//=============================================================================
// ST10_Flow22_JMagnetLifting.scl
// 1:1 CONVERSION FROM TIA PORTAL V18 GRAPH XML
// Generated: 2026-02-02
//=============================================================================

TYPE
    E_STEP_ST10_Flow22_JMagnetLifting : (
        STEP_ST10_Flow22_JMagnetLifting_WaitingPalletUnloading := 135,
        STEP_ST10_Flow22_JMagnetLifting_S3 := 3,
        STEP_ST10_Flow22_JMagnetLifting_TimeDelay := 22,
        STEP_ST10_Flow22_JMagnetLifting_J_magnetLiftingPalletLocationCylindertoHP := 129,
        STEP_ST10_Flow22_JMagnetLifting_Process_Finish := 237,
        STEP_ST10_Flow22_JMagnetLifting_F22_Initial := 1,
        STEP_ST10_Flow22_JMagnetLifting_S4 := 4,
        STEP_ST10_Flow22_JMagnetLifting_PalletRequest := 136,
        STEP_ST10_Flow22_JMagnetLifting_WaitRobotInitialFinish := 8,
        STEP_ST10_Flow22_JMagnetLifting_MotorCWStart := 24,
        STEP_ST10_Flow22_JMagnetLifting_J_magnetLiftingPalletLocationCylindertoHP_3 := 139,
        STEP_ST10_Flow22_JMagnetLifting_S2 := 2,
        STEP_ST10_Flow22_JMagnetLifting_RequestRobotPickPallet := 134,
        STEP_ST10_Flow22_JMagnetLifting_StatusError := 20,
        STEP_ST10_Flow22_JMagnetLifting_MotorCCWRun_1 := 144,
        STEP_ST10_Flow22_JMagnetLifting_CheckStopPalletExist := 21,
        STEP_ST10_Flow22_JMagnetLifting_MotorCCWStart := 23,
        STEP_ST10_Flow22_JMagnetLifting_S10_InitialFinish := 10,
        STEP_ST10_Flow22_JMagnetLifting_WaitRobotTaskFinish := 145,
        STEP_ST10_Flow22_JMagnetLifting_RobotCountClear0 := 137,
        STEP_ST10_Flow22_JMagnetLifting_MotorCCWRun := 140,
        STEP_ST10_Flow22_JMagnetLifting_J_magnetLiftingPalletLocationCylindertoHP_2 := 138,
        STEP_ST10_Flow22_JMagnetLifting_H_shaftLiftingLiftingCylinderToWP := 116,
        STEP_ST10_Flow22_JMagnetLifting_CheckPalletExist := 133,
        STEP_ST10_Flow22_JMagnetLifting_J_magnetLiftingPalletLocationCylindertoWP_1 := 130,
        STEP_ST10_Flow22_JMagnetLifting_Step131 := 131,
        STEP_ST10_Flow22_JMagnetLifting_CheckShaftLiftingCylinderPos := 117,
        STEP_ST10_Flow22_JMagnetLifting_J_magnetLiftingPalletLocationCylindertoHP_4 := 143,
        STEP_ST10_Flow22_JMagnetLifting_ProcessStart := 100,
        STEP_ST10_Flow22_JMagnetLifting_MotorStop := 132,
        STEP_ST10_Flow22_JMagnetLifting_Motor_Stop := 141,
        STEP_ST10_Flow22_JMagnetLifting_J_magnetLiftingCylinderToWP := 142,
        STEP_ST10_Flow22_JMagnetLifting_S5_MESInitial := 5,
    ) INT := 1;
END_TYPE

CONST
    STEP_ST10_Flow22_JMagnetLifting_WaitingPalletUnloading := 135;
    STEP_ST10_Flow22_JMagnetLifting_S3 := 3;
    STEP_ST10_Flow22_JMagnetLifting_TimeDelay := 22;
    STEP_ST10_Flow22_JMagnetLifting_J_magnetLiftingPalletLocationCylindertoHP := 129;
    STEP_ST10_Flow22_JMagnetLifting_Process_Finish := 237;
    STEP_ST10_Flow22_JMagnetLifting_F22_Initial := 1;
    STEP_ST10_Flow22_JMagnetLifting_S4 := 4;
    STEP_ST10_Flow22_JMagnetLifting_PalletRequest := 136;
    STEP_ST10_Flow22_JMagnetLifting_WaitRobotInitialFinish := 8;
    STEP_ST10_Flow22_JMagnetLifting_MotorCWStart := 24;
    STEP_ST10_Flow22_JMagnetLifting_J_magnetLiftingPalletLocationCylindertoHP_3 := 139;
    STEP_ST10_Flow22_JMagnetLifting_S2 := 2;
    STEP_ST10_Flow22_JMagnetLifting_RequestRobotPickPallet := 134;
    STEP_ST10_Flow22_JMagnetLifting_StatusError := 20;
    STEP_ST10_Flow22_JMagnetLifting_MotorCCWRun_1 := 144;
    STEP_ST10_Flow22_JMagnetLifting_CheckStopPalletExist := 21;
    STEP_ST10_Flow22_JMagnetLifting_MotorCCWStart := 23;
    STEP_ST10_Flow22_JMagnetLifting_S10_InitialFinish := 10;
    STEP_ST10_Flow22_JMagnetLifting_WaitRobotTaskFinish := 145;
    STEP_ST10_Flow22_JMagnetLifting_RobotCountClear0 := 137;
    STEP_ST10_Flow22_JMagnetLifting_MotorCCWRun := 140;
    STEP_ST10_Flow22_JMagnetLifting_J_magnetLiftingPalletLocationCylindertoHP_2 := 138;
    STEP_ST10_Flow22_JMagnetLifting_H_shaftLiftingLiftingCylinderToWP := 116;
    STEP_ST10_Flow22_JMagnetLifting_CheckPalletExist := 133;
    STEP_ST10_Flow22_JMagnetLifting_J_magnetLiftingPalletLocationCylindertoWP_1 := 130;
    STEP_ST10_Flow22_JMagnetLifting_Step131 := 131;
    STEP_ST10_Flow22_JMagnetLifting_CheckShaftLiftingCylinderPos := 117;
    STEP_ST10_Flow22_JMagnetLifting_J_magnetLiftingPalletLocationCylindertoHP_4 := 143;
    STEP_ST10_Flow22_JMagnetLifting_ProcessStart := 100;
    STEP_ST10_Flow22_JMagnetLifting_MotorStop := 132;
    STEP_ST10_Flow22_JMagnetLifting_Motor_Stop := 141;
    STEP_ST10_Flow22_JMagnetLifting_J_magnetLiftingCylinderToWP := 142;
    STEP_ST10_Flow22_JMagnetLifting_S5_MESInitial := 5;
END_CONST

FUNCTION_BLOCK "ST10_Flow22_JMagnetLifting_1to1"
{ S7_Optimized_Access := 'TRUE' }
VERSION : 1.0

VAR_INPUT
    iSysInface : "RCS_SysComInterface_V1";
END_VAR

VAR_IN_OUT
    ioPM_Inface : "RCS_PMInterface_V1";
    ioStatus : Int;
END_VAR

VAR_OUTPUT
    oAlarmID : Int;
END_VAR

VAR
    State : INT := 1;
    act_InitialRun : Bool;
    act_InitialOK : Bool;
    act_WaitRunning : Bool;
    act_Running : Bool;
    act_ProcessComplete : Bool;
    act_ProcessStart : Bool;
    act_UnPause : Bool;
    bError : Bool;
    wErrorID : Word;
END_VAR

BEGIN
    //======================================================================
    // STATE MACHINE - Inline Transition Conditions
    //======================================================================

    CASE #State OF

        // ===========================================
        // STEP 135: WaitingPalletUnloading
        // ===========================================
        STEP_ST10_Flow22_JMagnetLifting_WaitingPalletUnloading:
            // No actions in XML

            // Transition to next step: 3
            IF TRUE THEN  // Sequential transition - review XML for actual condition
                #State := STEP_ST10_Flow22_JMagnetLifting_S3;
            END_IF;

        // ===========================================
        // STEP 3: S3
        // ===========================================
        STEP_ST10_Flow22_JMagnetLifting_S3:
            // No actions in XML

            // Transition to next step: 22
            IF TRUE THEN  // Sequential transition - review XML for actual condition
                #State := STEP_ST10_Flow22_JMagnetLifting_TimeDelay;
            END_IF;

        // ===========================================
        // STEP 22: TimeDelay
        // ===========================================
        STEP_ST10_Flow22_JMagnetLifting_TimeDelay:
            // No actions in XML

            // Transition to next step: 129
            IF TRUE THEN  // Sequential transition - review XML for actual condition
                #State := STEP_ST10_Flow22_JMagnetLifting_J_magnetLiftingPalletLocationCylindertoHP;
            END_IF;

        // ===========================================
        // STEP 129: J-magnetLiftingPalletLocationCylindertoHP
        // ===========================================
        STEP_ST10_Flow22_JMagnetLifting_J_magnetLiftingPalletLocationCylindertoHP:
            // Action Qualifier=S
            // Token: "ST10Cylinder".Cy[32].Inout.AutoGoHome
            "ST10Cylinder".Cy[32].Inout.AutoGoHome := TRUE;
            // Action Qualifier=R
            // Token: "ST10Cylinder".Cy[32].Inout.AutoGoWork
            "ST10Cylinder".Cy[32].Inout.AutoGoWork := FALSE;

            // Transition to next step: 237
            IF TRUE THEN  // Sequential transition - review XML for actual condition
                #State := STEP_ST10_Flow22_JMagnetLifting_Process_Finish;
            END_IF;

        // ===========================================
        // STEP 237: Process Finish
        // ===========================================
        STEP_ST10_Flow22_JMagnetLifting_Process_Finish:
            // No actions in XML

            // Transition to next step: 1
            IF TRUE THEN  // Sequential transition - review XML for actual condition
                #State := STEP_ST10_Flow22_JMagnetLifting_F22_Initial;
            END_IF;

        // ===========================================
        // STEP 1: F22_Initial
        // ===========================================
        STEP_ST10_Flow22_JMagnetLifting_F22_Initial:
            // Action Qualifier=S
            // Token: #ioPM_Inface.InitialRun
            #ioPM_Inface.InitialRun := TRUE;
            // Action Qualifier=R
            // Token: #ioPM_Inface.InitialOK
            #ioPM_Inface.InitialOK := FALSE;
            // Action Qualifier=R
            // Token: #ioPM_Inface.WaitRunning
            #ioPM_Inface.WaitRunning := FALSE;
            // Action Qualifier=R
            // Token: #ioPM_Inface.Running
            #ioPM_Inface.Running := FALSE;
            // Action Qualifier=R
            // Token: #ioPM_Inface.ProcessComplete
            #ioPM_Inface.ProcessComplete := FALSE;
            // Action Qualifier=R
            // Token: #ioPM_Inface.UnPause
            #ioPM_Inface.UnPause := FALSE;
            // Action Qualifier=R
            // Token: "Station_Sys".Cmd.Calibration
            "Station_Sys".Cmd.Calibration := FALSE;
            // Action Qualifier=R
            // Token: "Station_Sys".Cmd.ChangeOver
            "Station_Sys".Cmd.ChangeOver := FALSE;
            // Action Qualifier=N
            // Token: //"ST350_Sys".Cmd.DryRun
            //"ST350_Sys".Cmd.DryRun;
            // Action Qualifier=R
            // Token: "Station_Sys".Cmd.Reserve
            "Station_Sys".Cmd.Reserve := FALSE;
            // Action Qualifier=R
            // Token: "Station_Sys".Cmd.OneCycle
            "Station_Sys".Cmd.OneCycle := FALSE;

            // Transition to next step: 4
            IF TRUE THEN  // Sequential transition - review XML for actual condition
                #State := STEP_ST10_Flow22_JMagnetLifting_S4;
            END_IF;

        // ===========================================
        // STEP 4: S4
        // ===========================================
        STEP_ST10_Flow22_JMagnetLifting_S4:
            // No actions in XML

            // Transition to next step: 136
            IF TRUE THEN  // Sequential transition - review XML for actual condition
                #State := STEP_ST10_Flow22_JMagnetLifting_PalletRequest;
            END_IF;

        // ===========================================
        // STEP 136: PalletRequest
        // ===========================================
        STEP_ST10_Flow22_JMagnetLifting_PalletRequest:
            // Action Qualifier=N
            // Token: "AutoProcessControl".Global.J.LoadStopRequestPallet_4
            "AutoProcessControl".Global.J.LoadStopRequestPallet_4;

            // Transition to next step: 8
            IF TRUE THEN  // Sequential transition - review XML for actual condition
                #State := STEP_ST10_Flow22_JMagnetLifting_WaitRobotInitialFinish;
            END_IF;

        // ===========================================
        // STEP 8: WaitRobotInitialFinish
        // ===========================================
        STEP_ST10_Flow22_JMagnetLifting_WaitRobotInitialFinish:
            // No actions in XML

            // Transition to next step: 24
            IF TRUE THEN  // Sequential transition - review XML for actual condition
                #State := STEP_ST10_Flow22_JMagnetLifting_MotorCWStart;
            END_IF;

        // ===========================================
        // STEP 24: MotorCWStart
        // ===========================================
        STEP_ST10_Flow22_JMagnetLifting_MotorCWStart:
            // Action Qualifier=R
            // Token: "MotorControl".Dev[2].Auto.CCWStart
            "MotorControl".Dev[2].Auto.CCWStart := FALSE;
            // Action Qualifier=S
            // Token: "MotorControl".Dev[2].Auto.Start
            "MotorControl".Dev[2].Auto.Start := TRUE;

            // Transition to next step: 139
            IF TRUE THEN  // Sequential transition - review XML for actual condition
                #State := STEP_ST10_Flow22_JMagnetLifting_J_magnetLiftingPalletLocationCylindertoHP_3;
            END_IF;

        // ===========================================
        // STEP 139: J-magnetLiftingPalletLocationCylindertoHP_3
        // ===========================================
        STEP_ST10_Flow22_JMagnetLifting_J_magnetLiftingPalletLocationCylindertoHP_3:
            // Action Qualifier=S
            // Token: "ST10Cylinder".Cy[31].Inout.AutoGoHome
            "ST10Cylinder".Cy[31].Inout.AutoGoHome := TRUE;
            // Action Qualifier=R
            // Token: "ST10Cylinder".Cy[31].Inout.AutoGoWork
            "ST10Cylinder".Cy[31].Inout.AutoGoWork := FALSE;

            // Transition to next step: 2
            IF TRUE THEN  // Sequential transition - review XML for actual condition
                #State := STEP_ST10_Flow22_JMagnetLifting_S2;
            END_IF;

        // ===========================================
        // STEP 2: S2
        // ===========================================
        STEP_ST10_Flow22_JMagnetLifting_S2:
            // No actions in XML

            // Transition to next step: 134
            IF TRUE THEN  // Sequential transition - review XML for actual condition
                #State := STEP_ST10_Flow22_JMagnetLifting_RequestRobotPickPallet;
            END_IF;

        // ===========================================
        // STEP 134: RequestRobotPickPallet
        // ===========================================
        STEP_ST10_Flow22_JMagnetLifting_RequestRobotPickPallet:
            // Action Qualifier=N
            // Token: "AutoProcessControl".J_MagnetLine.Robot2PickPrimit
            "AutoProcessControl".J_MagnetLine.Robot2PickPrimit;

            // Transition to next step: 20
            IF TRUE THEN  // Sequential transition - review XML for actual condition
                #State := STEP_ST10_Flow22_JMagnetLifting_StatusError;
            END_IF;

        // ===========================================
        // STEP 20: StatusError
        // ===========================================
        STEP_ST10_Flow22_JMagnetLifting_StatusError:
            // Action Qualifier=S
            // Token: "ST10_DeviceError".J.MagnetLine.LiftingCylStatusError
            "ST10_DeviceError".J.MagnetLine.LiftingCylStatusError := TRUE;

            // Transition to next step: 144
            IF TRUE THEN  // Sequential transition - review XML for actual condition
                #State := STEP_ST10_Flow22_JMagnetLifting_MotorCCWRun_1;
            END_IF;

        // ===========================================
        // STEP 144: MotorCCWRun_1
        // ===========================================
        STEP_ST10_Flow22_JMagnetLifting_MotorCCWRun_1:
            // Action Qualifier=S
            // Token: "MotorControl".Dev[2].Auto.CCWStart
            "MotorControl".Dev[2].Auto.CCWStart := TRUE;
            // Action Qualifier=S
            // Token: "MotorControl".Dev[2].Auto.Start
            "MotorControl".Dev[2].Auto.Start := TRUE;

            // Transition to next step: 21
            IF TRUE THEN  // Sequential transition - review XML for actual condition
                #State := STEP_ST10_Flow22_JMagnetLifting_CheckStopPalletExist;
            END_IF;

        // ===========================================
        // STEP 21: CheckStopPalletExist
        // ===========================================
        STEP_ST10_Flow22_JMagnetLifting_CheckStopPalletExist:
            // No actions in XML

            // Transition to next step: 23
            IF TRUE THEN  // Sequential transition - review XML for actual condition
                #State := STEP_ST10_Flow22_JMagnetLifting_MotorCCWStart;
            END_IF;

        // ===========================================
        // STEP 23: MotorCCWStart
        // ===========================================
        STEP_ST10_Flow22_JMagnetLifting_MotorCCWStart:
            // Action Qualifier=S
            // Token: "MotorControl".Dev[2].Auto.CCWStart
            "MotorControl".Dev[2].Auto.CCWStart := TRUE;
            // Action Qualifier=S
            // Token: "MotorControl".Dev[2].Auto.Start
            "MotorControl".Dev[2].Auto.Start := TRUE;

            // Transition to next step: 10
            IF TRUE THEN  // Sequential transition - review XML for actual condition
                #State := STEP_ST10_Flow22_JMagnetLifting_S10_InitialFinish;
            END_IF;

        // ===========================================
        // STEP 10: S10_InitialFinish
        // ===========================================
        STEP_ST10_Flow22_JMagnetLifting_S10_InitialFinish:
            // Action Qualifier=S
            // Token: #ioPM_Inface.InitialOK
            #ioPM_Inface.InitialOK := TRUE;

            // Transition to next step: 145
            IF TRUE THEN  // Sequential transition - review XML for actual condition
                #State := STEP_ST10_Flow22_JMagnetLifting_WaitRobotTaskFinish;
            END_IF;

        // ===========================================
        // STEP 145: WaitRobotTaskFinish
        // ===========================================
        STEP_ST10_Flow22_JMagnetLifting_WaitRobotTaskFinish:
            // No actions in XML

            // Transition to next step: 137
            IF TRUE THEN  // Sequential transition - review XML for actual condition
                #State := STEP_ST10_Flow22_JMagnetLifting_RobotCountClear0;
            END_IF;

        // ===========================================
        // STEP 137: RobotCountClear0
        // ===========================================
        STEP_ST10_Flow22_JMagnetLifting_RobotCountClear0:
            // Action Qualifier=N
            // Token: "KukaRobot2_CtrlDB".sPLCtoROB.User.Cycle.DI242_NewPallet
            "KukaRobot2_CtrlDB".sPLCtoROB.User.Cycle.DI242_NewPallet;
            // Action Qualifier=R
            // Token: "MotorControl".Dev[2].Auto.Start
            "MotorControl".Dev[2].Auto.Start := FALSE;

            // Transition to next step: 140
            IF TRUE THEN  // Sequential transition - review XML for actual condition
                #State := STEP_ST10_Flow22_JMagnetLifting_MotorCCWRun;
            END_IF;

        // ===========================================
        // STEP 140: MotorCCWRun
        // ===========================================
        STEP_ST10_Flow22_JMagnetLifting_MotorCCWRun:
            // Action Qualifier=S
            // Token: "MotorControl".Dev[2].Auto.CCWStart
            "MotorControl".Dev[2].Auto.CCWStart := TRUE;
            // Action Qualifier=S
            // Token: "MotorControl".Dev[2].Auto.Start
            "MotorControl".Dev[2].Auto.Start := TRUE;
            // Action Qualifier=R
            // Token: "MotorControl".Dev[14].Auto.CCWStart
            "MotorControl".Dev[14].Auto.CCWStart := FALSE;
            // Action Qualifier=S
            // Token: "MotorControl".Dev[14].Auto.Start
            "MotorControl".Dev[14].Auto.Start := TRUE;

            // Transition to next step: 138
            IF TRUE THEN  // Sequential transition - review XML for actual condition
                #State := STEP_ST10_Flow22_JMagnetLifting_J_magnetLiftingPalletLocationCylindertoHP_2;
            END_IF;

        // ===========================================
        // STEP 138: J-magnetLiftingPalletLocationCylindertoHP_2
        // ===========================================
        STEP_ST10_Flow22_JMagnetLifting_J_magnetLiftingPalletLocationCylindertoHP_2:
            // Action Qualifier=S
            // Token: "ST10Cylinder".Cy[32].Inout.AutoGoHome
            "ST10Cylinder".Cy[32].Inout.AutoGoHome := TRUE;
            // Action Qualifier=R
            // Token: "ST10Cylinder".Cy[32].Inout.AutoGoWork
            "ST10Cylinder".Cy[32].Inout.AutoGoWork := FALSE;

            // Transition to next step: 116
            IF TRUE THEN  // Sequential transition - review XML for actual condition
                #State := STEP_ST10_Flow22_JMagnetLifting_H_shaftLiftingLiftingCylinderToWP;
            END_IF;

        // ===========================================
        // STEP 116: H-shaftLiftingLiftingCylinderToWP
        // ===========================================
        STEP_ST10_Flow22_JMagnetLifting_H_shaftLiftingLiftingCylinderToWP:
            // Action Qualifier=R
            // Token: "ST10Cylinder".Cy[31].Inout.AutoGoHome
            "ST10Cylinder".Cy[31].Inout.AutoGoHome := FALSE;
            // Action Qualifier=S
            // Token: "ST10Cylinder".Cy[31].Inout.AutoGoWork
            "ST10Cylinder".Cy[31].Inout.AutoGoWork := TRUE;

            // Transition to next step: 133
            IF TRUE THEN  // Sequential transition - review XML for actual condition
                #State := STEP_ST10_Flow22_JMagnetLifting_CheckPalletExist;
            END_IF;

        // ===========================================
        // STEP 133: CheckPalletExist
        // ===========================================
        STEP_ST10_Flow22_JMagnetLifting_CheckPalletExist:
            // No actions in XML

            // Transition to next step: 130
            IF TRUE THEN  // Sequential transition - review XML for actual condition
                #State := STEP_ST10_Flow22_JMagnetLifting_J_magnetLiftingPalletLocationCylindertoWP_1;
            END_IF;

        // ===========================================
        // STEP 130: J-magnetLiftingPalletLocationCylindertoWP_1
        // ===========================================
        STEP_ST10_Flow22_JMagnetLifting_J_magnetLiftingPalletLocationCylindertoWP_1:
            // Action Qualifier=R
            // Token: "ST10Cylinder".Cy[32].Inout.AutoGoHome
            "ST10Cylinder".Cy[32].Inout.AutoGoHome := FALSE;
            // Action Qualifier=S
            // Token: "ST10Cylinder".Cy[32].Inout.AutoGoWork
            "ST10Cylinder".Cy[32].Inout.AutoGoWork := TRUE;

            // Transition to next step: 131
            IF TRUE THEN  // Sequential transition - review XML for actual condition
                #State := STEP_ST10_Flow22_JMagnetLifting_Step131;
            END_IF;

        // ===========================================
        // STEP 131: Step131
        // ===========================================
        STEP_ST10_Flow22_JMagnetLifting_Step131:
            // No actions in XML

            // Transition to next step: 117
            IF TRUE THEN  // Sequential transition - review XML for actual condition
                #State := STEP_ST10_Flow22_JMagnetLifting_CheckShaftLiftingCylinderPos;
            END_IF;

        // ===========================================
        // STEP 117: CheckShaftLiftingCylinderPos
        // ===========================================
        STEP_ST10_Flow22_JMagnetLifting_CheckShaftLiftingCylinderPos:
            // No actions in XML

            // Transition to next step: 143
            IF TRUE THEN  // Sequential transition - review XML for actual condition
                #State := STEP_ST10_Flow22_JMagnetLifting_J_magnetLiftingPalletLocationCylindertoHP_4;
            END_IF;

        // ===========================================
        // STEP 143: J-magnetLiftingPalletLocationCylindertoHP_4
        // ===========================================
        STEP_ST10_Flow22_JMagnetLifting_J_magnetLiftingPalletLocationCylindertoHP_4:
            // Action Qualifier=S
            // Token: "ST10Cylinder".Cy[32].Inout.AutoGoHome
            "ST10Cylinder".Cy[32].Inout.AutoGoHome := TRUE;
            // Action Qualifier=R
            // Token: "ST10Cylinder".Cy[32].Inout.AutoGoWork
            "ST10Cylinder".Cy[32].Inout.AutoGoWork := FALSE;

            // Transition to next step: 100
            IF TRUE THEN  // Sequential transition - review XML for actual condition
                #State := STEP_ST10_Flow22_JMagnetLifting_ProcessStart;
            END_IF;

        // ===========================================
        // STEP 100: ProcessStart
        // ===========================================
        STEP_ST10_Flow22_JMagnetLifting_ProcessStart:
            // Action Qualifier=R
            // Token: #ioPM_Inface.InitialRun
            #ioPM_Inface.InitialRun := FALSE;
            // Action Qualifier=R
            // Token: #ioPM_Inface.ProcessComplete
            #ioPM_Inface.ProcessComplete := FALSE;
            // Action Qualifier=R
            // Token: #ioPM_Inface.ProcessStart
            #ioPM_Inface.ProcessStart := FALSE;
            // Action Qualifier=S
            // Token: #ioPM_Inface.InitialOK
            #ioPM_Inface.InitialOK := TRUE;
            // Action Qualifier=S
            // Token: #ioPM_Inface.WaitRunning
            #ioPM_Inface.WaitRunning := TRUE;
            // Action Qualifier=N, Event="S1"
            // Token: #ioPM_Inface.ProcessResult := 0
            #ioPM_Inface.ProcessResult := 0;
            // Action Qualifier=R
            // Token: "ST10_GeneralData".FlowControl_Handshake[21].Start
            "ST10_GeneralData".FlowControl_Handshake[21].Start := FALSE;
            // Action Qualifier=R
            // Token: "ST10_GeneralData".FlowControl_Handshake[21].Done
            "ST10_GeneralData".FlowControl_Handshake[21].Done := FALSE;
            // Action Qualifier=R
            // Token: "MotorControl".Dev[2].Auto.CCWStart
            "MotorControl".Dev[2].Auto.CCWStart := FALSE;
            // Action Qualifier=R
            // Token: "MotorControl".Dev[2].Auto.Start
            "MotorControl".Dev[2].Auto.Start := FALSE;

            // Transition to next step: 132
            IF TRUE THEN  // Sequential transition - review XML for actual condition
                #State := STEP_ST10_Flow22_JMagnetLifting_MotorStop;
            END_IF;

        // ===========================================
        // STEP 132: MotorStop
        // ===========================================
        STEP_ST10_Flow22_JMagnetLifting_MotorStop:
            // Action Qualifier=R
            // Token: "MotorControl".Dev[2].Auto.CCWStart
            "MotorControl".Dev[2].Auto.CCWStart := FALSE;
            // Action Qualifier=R
            // Token: "MotorControl".Dev[2].Auto.Start
            "MotorControl".Dev[2].Auto.Start := FALSE;

            // Transition to next step: 141
            IF TRUE THEN  // Sequential transition - review XML for actual condition
                #State := STEP_ST10_Flow22_JMagnetLifting_Motor_Stop;
            END_IF;

        // ===========================================
        // STEP 141: Motor Stop
        // ===========================================
        STEP_ST10_Flow22_JMagnetLifting_Motor_Stop:
            // Action Qualifier=R
            // Token: "MotorControl".Dev[2].Auto.CCWStart
            "MotorControl".Dev[2].Auto.CCWStart := FALSE;
            // Action Qualifier=R
            // Token: "MotorControl".Dev[2].Auto.Start
            "MotorControl".Dev[2].Auto.Start := FALSE;

            // Transition to next step: 142
            IF TRUE THEN  // Sequential transition - review XML for actual condition
                #State := STEP_ST10_Flow22_JMagnetLifting_J_magnetLiftingCylinderToWP;
            END_IF;

        // ===========================================
        // STEP 142: J-magnetLiftingCylinderToWP
        // ===========================================
        STEP_ST10_Flow22_JMagnetLifting_J_magnetLiftingCylinderToWP:
            // Action Qualifier=R
            // Token: "ST10Cylinder".Cy[31].Inout.AutoGoHome
            "ST10Cylinder".Cy[31].Inout.AutoGoHome := FALSE;
            // Action Qualifier=S
            // Token: "ST10Cylinder".Cy[31].Inout.AutoGoWork
            "ST10Cylinder".Cy[31].Inout.AutoGoWork := TRUE;

            // Transition to next step: 5
            IF TRUE THEN  // Sequential transition - review XML for actual condition
                #State := STEP_ST10_Flow22_JMagnetLifting_S5_MESInitial;
            END_IF;

        // ===========================================
        // STEP 5: S5_MESInitial
        // ===========================================
        STEP_ST10_Flow22_JMagnetLifting_S5_MESInitial:
            // No actions in XML

    END_CASE;

    // UPDATE ioPM_Inface
    #ioPM_Inface.InitialRun := #act_InitialRun;
    #ioPM_Inface.InitialOK := #act_InitialOK;
    #ioPM_Inface.WaitRunning := #act_WaitRunning;
    #ioPM_Inface.Running := #act_Running;
    #ioPM_Inface.ProcessComplete := #act_ProcessComplete;
    #ioPM_Inface.ProcessStart := #act_ProcessStart;
    #ioPM_Inface.UnPause := #act_UnPause;

    // ERROR HANDLING
    IF #bError THEN
        #ioStatus := 900;
        #oAlarmID := INT_TO_WORD(#wErrorID);
    ELSE
        #ioStatus := 0;
        #oAlarmID := 0;
    END_IF;
END_FUNCTION_BLOCK

//=============================================================================
// END OF FILE
//=============================================================================
